// TwinCAT 3 PLC project Main
// ProgramVersion: 3.1.4024.0
// libraries:
//   mobject-core, * (mobject)
//   mobject-graph, * (mobject)
//   mobject-graph-plc-pack, * (mobject)
//   mobject-graph-vision-pack, * (mobject)
//   mobject-server, * (mobject)
//   Tc2_Standard, * (Beckhoff Automation GmbH)
//   Tc2_System, * (Beckhoff Automation GmbH)
//   Tc2_Utilities, * (Beckhoff Automation GmbH)
//   Tc3_Module, * (Beckhoff Automation GmbH)
//   Tc3_Vision, * (Beckhoff Automation GmbH)
// project tree:
//   / PlcTask.TcTTO (not stored)
//   POUs/Examples/ MyCustomNode.TcPOU (not stored)
//   POUs/ MAIN.TcPOU
// real-time tasks:
//   TASK PlcTask: cycle T#10ms, priority 20, ADS port 350

// ---- POUs/MAIN.TcPOU
PROGRAM MAIN
VAR		

	// installation of the packs is only requried once. 
	initialise: BOOL;
	
	// graph packs
	iecDatatypesPack : IecDatatypesPack; // mobject-graph, 
	plcPack : PlcPack; // mobject-graph-plc-pack
	visionPack : VisionPack; // mobject-graph-vision-pack
	
	// custom node
	myCustomNode : MyCustomNode;

	// application
	graphFramework : GraphFramework;
	server : RpcServer;
	graphFrameworkApi : GraphFrameworkApi(graphFramework);	

END_VAR

IF NOT initialise THEN

	// add graph packs here...
	graphFramework.Install(iecDatatypesPack); // adds primitives such as BOOL, WORD, STRING...
	graphFramework.Install(plcPack); // adds datatypes and nodes base on TC2_Utilities...
	graphFramework.Install(visionPack); // adds datatypes and nodes for TC3_Vision...
	
	// add any custom datatypes here...
	// graphFramework.Datatypes.RegisterDatatype(_customDatatype);
	
	// add any custom nodes here...
	graphFramework.NodeFactory.AddNodeAsPrototype('Custom/MyCustomNode', myCustomNode);
	
	// add the graph framework api to the server, this will register all of the endpoint handlers
	server.RegisterApi(graphFrameworkApi);

	// done
	initialise := TRUE;	

END_IF

// a special feature of .RegisterApi is that the server will know to cyclic call all registered apis each cycle. 
server.CyclicCall();

END_PROGRAM
